{attribute 'linkalways'} 
{attribute 'no_explicit_call' := 'This FB is a CLASS and must be accessed using methods or properties'}
{attribute 'enable_dynamic_creation'}
FUNCTION_BLOCK _BIT EXTENDS DatatypeBase implements I_BitDatatype
VAR
	initialised : BOOL;
	activeParent : I_StructuredDatatype;
	activeByteOffset : PVOID;
	activeBitOffset : DWORD;
END_VAR

PROPERTY PUBLIC Address : PVOID
GET
IF NOT initialised THEN 
	RETURN;
END_IF

Address := activeParent.Address + activeByteOffset;
END_GET
END_PROPERTY

PROPERTY PUBLIC BitOffset : DWORD
GET
IF NOT initialised THEN 
	RETURN;
END_IF

BitOffset := activeBitOffset;
END_GET
END_PROPERTY

PROPERTY PUBLIC ByteOffset : PVOID
GET
IF NOT initialised THEN 
	RETURN;
END_IF

ByteOffset := activeByteOffset;
END_GET
END_PROPERTY

METHOD PUBLIC ClearReference
VAR_INPUT
END_VAR
activeParent := 0;
activeByteOffset := 0;
activeBitOffset := 0;
initialised := FALSE;
END_METHOD

METHOD PUBLIC Clone : I_Datatype
VAR
    pClone : POINTER TO _BIT;
END_VAR
pClone := __NEW(_BIT);

IF initialised THEN
	pClone^.MakeReferenceTo(activeParent, activeByteOffset, activeBitOffset);
END_IF

Clone := pClone^;
END_METHOD

METHOD PRIVATE GetBitValue : BOOL
VAR
	pByte : POINTER TO BYTE := Address;
END_VAR
IF NOT initialised THEN
	RETURN;
END_IF

CASE activeBitOffset OF
	0: GetBitValue := pByte^.0;
	1: GetBitValue := pByte^.1;
	2: GetBitValue := pByte^.2;
	3: GetBitValue := pByte^.3;
	4: GetBitValue := pByte^.4;
	5: GetBitValue := pByte^.5;
	6: GetBitValue := pByte^.6;
	7: GetBitValue := pByte^.7;
END_CASE;
END_METHOD

METHOD PUBLIC MakeReferenceTo
VAR_INPUT
	Parent : I_StructuredDatatype;
	ByteOffset : PVOID;
	BitOffset : DWORD;
END_VAR
activeParent := Parent;
activeByteOffset := ByteOffset;
activeBitOffset := BitOffset AND 16#7;
initialised := TRUE;
END_METHOD

PROPERTY PUBLIC Parent : I_StructuredDatatype
GET
Parent := activeParent;
END_GET
END_PROPERTY

METHOD PUBLIC SerializeWith
VAR_INPUT
	Serializer : I_Serializer;
END_VAR
Serializer.AddBool(GetBitValue());
END_METHOD

METHOD PRIVATE SetBitValue : BOOL
VAR_INPUT
	Value : BOOL;
END_VAR
VAR
	pByte : POINTER TO BYTE := Address;
END_VAR
IF NOT initialised THEN
	RETURN;
END_IF

CASE activeBitOffset OF
	0: pByte^.0 := Value;
	1: pByte^.1 := Value;
	2: pByte^.2 := Value;
	3: pByte^.3 := Value;
	4: pByte^.4 := Value;
	5: pByte^.5 := Value;
	6: pByte^.6 := Value;
	7: pByte^.7 := Value;
END_CASE;
END_METHOD

PROPERTY PUBLIC Size : UDINT
GET
Size := 1;
END_GET
END_PROPERTY

METHOD TryDeserializeFrom : BOOL
VAR_INPUT
	Deserializer : I_Deserializer;
	Feedback : I_DeserializerFeedback;
END_VAR
VAR 
	value : BOOL;
END_VAR
IF NOT Deserializer.TryGetBool(value, Feedback) THEN
	RETURN;
END_IF

SetBitValue(value);
TryDeserializeFrom := TRUE;
END_METHOD

METHOD TryMakeReferenceTo : BOOL
VAR_INPUT
	Target : I_Datatype;
END_VAR
VAR
	targetAsBit : I_BitDatatype;
END_VAR
IF NOT Target.TryResolveAsBitDatatype(targetAsBit) THEN
	RETURN;
END_IF

MakeReferenceTo(targetAsBit.Parent, targetAsBit.ByteOffset, targetAsBit.BitOffset);
TryMakeReferenceTo := TRUE;
END_METHOD

METHOD PUBLIC TryResolveAsBitDatatype : BOOL
VAR_INPUT
	Destination : REFERENCE TO I_BitDatatype;
END_VAR
Destination := this^;
TryResolveAsBitDatatype := TRUE;
END_METHOD

PROPERTY PUBLIC TypeName : T_MAXSTRING
GET
TypeName := 'BIT';
END_GET
END_PROPERTY

PROPERTY PUBLIC Value : BOOL
GET
Value := GetBitValue();
END_GET
SET
SetBitValue(Value);
END_SET
END_PROPERTY

END_FUNCTION_BLOCK

(* stored: Version 1.1.0.1, ProductVersion 3.1.4024.12
   POU _BIT: Id {d1424362-55ba-4d92-a95d-e8783b2964a0}, SpecialFunc None
   Folder Private: Id {c3d05154-870e-475c-a27e-cd1fcffe3cf1}
   Property Address: Id {8ce2401c-05df-4eb1-aaaa-e51cf82b4182}
   Get Get: Id {545c811f-eef1-45c7-a4ab-f506d6cb452d}
   Property BitOffset: Id {735eba2b-20b5-4bf7-9f38-96a145fea705}
   Get Get: Id {0a2641ac-3657-4e69-9fac-22f8de72fc1f}
   Property ByteOffset: Id {d1b6fa75-0c02-49b9-bb4e-aabb416fdfae}
   Get Get: Id {d9f7ed97-5e68-43fa-a0fa-97a8e00d3dda}
   Method ClearReference: Id {5c376c4e-accf-4f1a-bb6d-379d0cfc8b00}
   Method Clone: Id {753ceb0f-b2bc-448c-b8ee-6f5ba0d1bb9c}
   Method GetBitValue: Id {e718f332-2d9f-4470-bca6-2e66196e89da}
   Method MakeReferenceTo: Id {02d8f63e-1347-43cf-906d-8d5aad1dd547}
   Property Parent: Id {4f72d0f5-a246-4460-b19a-3ed250554bc0}
   Get Get: Id {27048d9f-42bf-4f72-8544-b8a04c1b55bf}
   Method SerializeWith: Id {baca04a6-9a00-45e4-9c70-c5893a3fbacb}
   Method SetBitValue: Id {eb7119ad-8b00-47f4-93cf-15e68d899c91}
   Property Size: Id {2d097b90-a037-4e11-98c2-b872aed4fe5c}
   Get Get: Id {6f6242e3-ce9b-4842-95d3-8b6375c06015}
   Method TryDeserializeFrom: Id {7f223bf3-10e0-4d0f-90c0-9e425c9e8a7e}
   Method TryMakeReferenceTo: Id {885b2714-b6a4-48c4-8eed-f9f3bcd35447}
   Method TryResolveAsBitDatatype: Id {19d25133-7123-4fdb-9973-911d4285cbcc}
   Property TypeName: Id {01e01daf-5c20-4c7e-9e2f-d72201aed978}
   Get Get: Id {372186b1-53af-4265-bca2-ff200db394a0}
   Property Value: Id {ec906a72-0494-4dde-a569-fe54fde95591}
   Get Get: Id {109c7b57-8357-40aa-a6ff-805ba5ee1838}
   Set Set: Id {fa60ea83-5f75-4446-908d-6f3bf2f111bb} *)
